// TIA Portal V16 export
// export: Created 2023-08-28T09:37:32.3577753Z, ExportSetting WithDefaults, DisplayName Totally Integrated Automation Portal, DisplayVersion V16 Update 6, DisplayName TIA Portal Version Control Interface, DisplayVersion V16 Update 2, DisplayName TIA Portal Openness, DisplayVersion V16 Update 6, DisplayName STEP 7 Professional, DisplayVersion V16 Update 6, DisplayName STEP 7 Safety, DisplayVersion V16, DisplayName WinCC Advanced, DisplayVersion V16 Update 6
FUNCTION_BLOCK "01_E_cleaning_the_alarm_reset_button"   // FB32, LAD
TITLE = cleaning the alarm reset button
{ S7_Optimized_Access := 'TRUE' }
AUTHOR : rtecme
VERSION : 0.1
// Funkcja resetuje znacznik ustawiany z HMI służący do kasowania alarów ekranów
// stored: AutoNumber true, IsIECCheckEnabled false, IsRetainMemResEnabled false, MemoryReserve 100, SetENOAutomatically false, UDAEnableTagReadback false
BEGIN

REGION Network 1: Reset Bitu Kasowania Alarmów
   // Po wykonaniu kasowania alarmów bit -0 jest zerowany
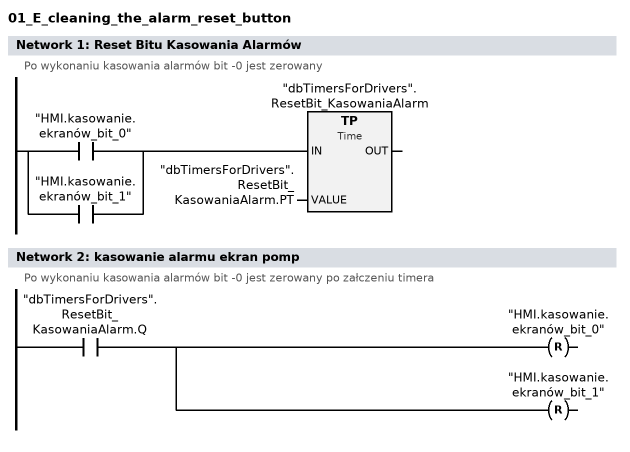
   "dbTimersForDrivers".ResetBit_KasowaniaAlarm.TP(IN := "HMI.kasowanie.ekranów_bit_0" OR "HMI.kasowanie.ekranów_bit_1", PT := "dbTimersForDrivers".ResetBit_KasowaniaAlarm.PT);   // TP coil
END_REGION

REGION Network 2: kasowanie alarmu ekran pomp
   // Po wykonaniu kasowania alarmów bit -0 jest zerowany po załczeniu timera
   RUNG wire#powerrail
      Contact( "dbTimersForDrivers".ResetBit_KasowaniaAlarm.Q )
      wire#w1
      R_Coil( "HMI.kasowanie.ekranów_bit_0" )
   END_RUNG
   RUNG wire#w1
      R_Coil( "HMI.kasowanie.ekranów_bit_1" )
   END_RUNG
   // the same network as SCL:
   IF "dbTimersForDrivers".ResetBit_KasowaniaAlarm.Q THEN
       "HMI.kasowanie.ekranów_bit_0" := FALSE;
       "HMI.kasowanie.ekranów_bit_1" := FALSE;
   END_IF;
END_REGION
END_FUNCTION_BLOCK
